INTERFACE ITcoManageable EXTENDS ITcoObject

METHOD RegisterManager : BOOL
VAR_INPUT
	Manager	:	ITcoObject;
END_VAR
END_METHOD

METHOD UnregisterManager : BOOL
VAR_INPUT
	Manager	:	ITcoObject;
END_VAR
END_METHOD

END_INTERFACE

(* stored: Version 1.1.0.1, ProductVersion 3.1.4024.6
   Itf ITcoManageable: Id {7897508a-1bfc-0e91-1dcb-4d0926cb3304}
   Method RegisterManager: Id {65512763-d28a-0764-0e23-4005c37574f7}
   Method UnregisterManager: Id {67f56503-47d4-0bd6-08ee-f8c089efb06d} *)
